// Some aggregate that has implemented a timer for demonstration.
FUNCTION_BLOCK FB_TimerAggregateA EXTENDS FB_BA_AggregateA
VAR_OUTPUT
	bOpen			: BOOL;
END_VAR
VAR
	Delay			: TON					:= (PT:=T#25S);
END_VAR

SUPER^();

Delay(IN := (bActiveEn AND (fActiveVal > 0.0)));
bOpen := Delay.Q;

END_FUNCTION_BLOCK

(* stored: Version 1.1.0.1, ProductVersion 3.1.4024.5
   POU FB_TimerAggregateA: Id {a1e3767a-21ef-4020-8623-53d1c21d6066}, SpecialFunc None *)
